// Methods for traversing a binary search tree.
{attribute 'qualified_only'}
{attribute 'to_string'}
TYPE E_BINARY_SEARCH_TREE_TRAVERSAL :
(
	In_Order := 0,
	Pre_Order,
	Post_Order, 
	Level_Order
)BYTE;
END_TYPE

(* stored: Version 1.1.0.1, ProductVersion 3.1.4024.4
   EnumerationTextList E_BINARY_SEARCH_TREE_TRAVERSAL: Id {3e0edefa-b709-0855-345d-bee12ed26c98} *)
